(* obsolete support after version 2.7.0.1
-------------------------read the document bellow---------------------------------------------------------------*)
FUNCTION_BLOCK FB_IPRO_ModbusRTU EXTENDS FB_ModbusSlaveRtu IMPLEMENTS I_Ipro_MotorPower;
VAR
	eState : E_AxisState;
// Write Modbus
	bControlModeSwitchCommand	: BOOL;						(* write p4.15 *)
	bFieldbusEnableServoCommand	:  BOOL;					(* write p4.11 0:Disable, 1:Anable *)
	eControlMode : E_IProCtrlMode;
	lrPositivePositionSoftwareLimit : LREAL;
	lrNagativePositionSoftwareLimit	: LREAL;
	lrMaxSpeedLimitOfControlModeSwitch : LREAL := 100;		(* P0.90 Add:1180 :Set the max. running speed during positioning when switching from speed mode or torque mode to position mode under position/speed, position/torque compound mode.*)
	lrPositionCmd : LREAL;									(* p4.12 Position value unit:(10000/rotary) *)
	lrSpeedCmd : LREAL;										(* p4.13 Unit:(rotary/minute) *)
	lrTorqueCmd	: LREAL; 									(* p4.14 Unit:% *)
	lrMaxSpeed	: LREAL; 									(* p4.31 Unit:(rotary/minute) *)
	lrMaxTorque	: LREAL; 									(* p0.10 Unit:% *) 
	bEmergenCyStop : BOOL;									(* p4.23 add:1846 16 bit :If P4.10 is 1, this parameter can be used to set emergency stop command. *)
	
// Read modbus
	lrSpeedFeedback	: LREAL;								(* r0.00 *) 
	lrTorqueFeedback : LREAL;								(* r0.06 *)
	lrPositionFeedback : LREAL;								(* r0.02 *)
	nFaultCode : INT; 										(* r0.99 *)
	eSystemStatus : E_IProStatus; 							(* r0.30 *)
	eCurrentMode : E_IProCurrentMode ;						(* r0.32 0: Position mode, 1: speed mode, 2: torque Mode*) 
							
	TempData_Word2real : U_Word2Real;
	TempData_Word2Dint	: U_Word2Dint;
	TempData_Word2Int	: U_Word2Int;

// State Handing
	bInit: BOOL;
	bHome: BOOL;
	bBusy: BOOL;
	bMoveAbsolute: BOOL;
	bReset: BOOL;
	bMoveTorque: BOOL;
	bStopped: BOOL; 						// StopDone
	bStop: BOOL;							// StopRequest
	lrHomePosition: LREAL;
	bHomed: BOOL;							// home done
	bInited: BOOL;							// Init Done
	bMoveAbsoluted: BOOL;					// MoveAbs Done
	bMoveTorqued: BOOL;						// MoveTorque Done
	bAbort: BOOL;							// Abort Request
	bActive: BOOL;
END_VAR

(*-------------------Document-------------
	1 set param in drive soft
	2 if set the control mode is different than Curren control mode on the Drive, The drive need restart by drive soft OR turn off power
	3 if the control mode swith command is TRUE, the current control mode will change according to the second mode if eControlMode have
	for example eControlMode = PositionTorque, when bControlModeSwitchCommand = false , currentmode is Position, else current mode is torque if it can
*)

bActive := eState >= AXIS_READY_INITIALIZED;
StateMachine();
bError := nFaultCode <> 0;
SUPER^();
CASE eState OF
	AXIS_INITIALIZING..AXIS_RESET_DONE, AXIS_ABORTING:
		tonConfirmReallyError(
			IN := bError OR bModbusError,
			PT := timeConfirmReallyError,
			Q => bReallyError 
		);
END_CASE

PROPERTY Active : bool
GET
Active := bActive;
END_GET
END_PROPERTY

{attribute 'monitoring' := 'variable'}
PROPERTY Busy : bool
GET
Busy := bBusy;
END_GET
END_PROPERTY

PROPERTY ControlMode : E_IProCtrlMode
GET
END_GET
SET
IF eState = AXIS_UNINITIALIZED THEN
	THIS^.eControlMode := ControlMode;
END_IF
END_SET
END_PROPERTY

PROPERTY ControlModeSwitchCmd : bool
GET
ControlModeSwitchCmd := bControlModeSwitchCommand;
END_GET
END_PROPERTY

METHOD Convert : BOOL
VAR_INPUT
	iRegionNo	:	INT;
	pReadData	:	POINTER TO word;
END_VAR
VAR
	iLoop		: 	INT;
	TempData	:	 U_Word2Dint;
	TempData_w2i	: U_Word2Int;
	TempData_Int	: INT;
END_VAR
	TempData.iWord[0] := pReadData[0];
	TempData.iWord[1] := pReadData[1];
	TempData_w2i.iWord := pReadData[0];
	TempData_Int := TempData_w2i.iInt;
CASE iRegionNo OF 
	0:// speed 0.1 r/m
		lrSpeedFeedback := DINT_TO_LREAL(TempData.idInt)*0.1;//32 bit
	1:// position unit 1
	
		lrPositionFeedback := DINT_TO_LREAL(TempData.idInt); //64 bit
	2:// torque 0.1
		lrTorqueFeedback := INT_TO_LREAL(TempData_Int)*0.1;
	3:
		eSystemStatus := pReadData[0];
	4:
		eCurrentMode := pReadData[0];
	5:
		nFaultCode := pReadData[0];// must not use word to int

	
END_CASE
END_METHOD

PROPERTY CurrentMode : E_IProCurrentMode
GET
CurrentMode := eCurrentMode;
END_GET
END_PROPERTY

PROPERTY Enable : bool
GET
Enable := bFieldbusEnableServoCommand;
END_GET
END_PROPERTY

PROPERTY ErrorID : REFERENCE TO INT
GET
ErrorID REF= nFaultCode;
END_GET
END_PROPERTY

{attribute 'monitoring' := 'variable'}
PROPERTY InPosition : bool
GET
InPosition := F_CheckInRange( lrHighLimit := lrPositionFeedback + 20,
						lrLowLimit := lrPositionFeedback - 20,
						lrValue := lrPositionCmd)	;
END_GET
END_PROPERTY

PROPERTY IsHomed : bool
GET
IsHomed := F_CheckInRange( lrHighLimit := lrPositionFeedback + 10,
						lrLowLimit := lrPositionFeedback - 10,
						lrValue := lrHomePosition)	;
END_GET
END_PROPERTY

PROPERTY IsInTorque : bool
GET
isIntorque := F_CheckInRange( lrHighLimit := lrTorqueFeedback + 0.5,// 1%
					lrLowLimit := lrTorqueFeedback -0.5 ,
					lrValue := lrTorqueCmd) ;// +-0.5%	;
END_GET
END_PROPERTY

PROPERTY IsStop : bool // not moving
GET
IsStop := eSystemStatus = IPRO_STATUS_FAULT;
END_GET
END_PROPERTY

PROPERTY MaxSpeed : lreal// large than 0
GET
MaxSpeed := lrMaxSpeed;
END_GET
SET
IF eState = AXIS_UNINITIALIZED THEN
	lrMaxSpeed := MaxSpeed;
END_IF
END_SET
END_PROPERTY

PROPERTY MaxTorque : Lreal// // % larger than 0
GET
MaxTorque := lrMaxTorque;
END_GET
SET
IF eState = AXIS_UNINITIALIZED THEN
	lrMaxTorque := MaxTorque;
END_IF

arrAddressWrite[10][2] :=  LREAL_TO_WORD(ABS(lrMaxTorque*10));
END_SET
END_PROPERTY

METHOD MR_Abort : BOOL // THIS IS REQUEST ABORT. => ACTIVE = False
IF eState >= AXIS_INITIALIZING THEN
	bAbort := TRUE;
	MR_Abort := FALSE;
	bBusy := TRUE;
	eState := AXIS_ABORTING;
ELSIF eState = AXIS_UNINITIALIZED THEN
	bAbort := FALSE;
	MR_Abort := TRUE;
	bBusy := False;
END_IF
END_METHOD

METHOD MR_Home : BOOL // control mode must have Position Mode // actually it the same as MOVE absolute 
VAR_INPUT
	lrHomePosition : LREAL;
END_VAR
IF eState = AXIS_IDLE AND eCurrentMode = IPRO_CURRENT_MODE_POSITION 
AND NOT F_CheckInRange(lrHighLimit := lrHomePosition + 10,
					lrLowLimit := lrHomePosition - 10,
					lrValue := lrPositionFeedback)
THEN 
	bHome := TRUE;
	bHomed := FALSE;
	bBusy := TRUE;
	MR_Home := FALSE;
 	eState := AXIS_HOME;
	THIS^.lrHomePosition := lrHomePosition;
ELSIF  eState = AXIS_IDLE AND eCurrentMode <> IPRO_CURRENT_MODE_POSITION THEN 
	bHome := TRUE;
	bHomed := FALSE;
	bBusy := TRUE;
	MR_Home := FALSE;
 	MS_SwitchMode(eModeChangeTo := IPRO_CURRENT_MODE_POSITION);

ELSIF eState = AXIS_HOME_DONE THEN
	bHomed := TRUE;
	bHome := FALSE;
	bBusy := FALSE;
	MR_Home := TRUE;
END_IF
END_METHOD

METHOD MR_Init : BOOL
IF eState = AXIS_UNINITIALIZED THEN
	bInit := TRUE;
	bInited := FALSE;
	bBusy := TRUE;
	MR_Init := FALSE;
	eState := AXIS_INITIALIZING;
ELSIF eState = AXIS_READY_INITIALIZED THEN
	bInited := True;
	bInit := FALSE;
	bBusy := FALSE;
	MR_Init := TRUE;
	
END_IF
END_METHOD

METHOD MR_MoveAbsolute : BOOL // control mode must have Position Mode
VAR_INPUT
	lrAbsolutePosition : LREAL;
END_VAR
IF eState = AXIS_IDLE 
AND eCurrentMode = IPRO_CURRENT_MODE_POSITION 
AND NOT F_CheckInRange( lrHighLimit := lrPositionFeedback + 10,
						lrLowLimit := lrPositionFeedback - 10,
						lrValue := lrAbsolutePosition)													
THEN
	lrPositionCmd := lrAbsolutePosition;
	MR_MoveAbsolute := FALSE;
	bBusy := TRUE;
	bMoveAbsolute := TRUE;
	bMoveAbsoluted := FALSE;
	eState := AXIS_MOVE_ABSOLUTE;
ELSIF eState = AXIS_IDLE  AND eCurrentMode <> IPRO_CURRENT_MODE_POSITION THEN
	MR_MoveAbsolute := FALSE;
	bBusy := TRUE;
	bMoveAbsolute := TRUE;
	bMoveAbsoluted := FALSE;
	MS_SwitchMode( eModeChangeTo := IPRO_CURRENT_MODE_POSITION);// if switch mode ok => eCurrentMode = AXIS_CURRENT_MODE_POSITION 

ELSIF eState = AXIS_MOVE_ABSOLUTE_DONE THEN
	bBusy := FALSE;
	bMoveAbsolute := FALSE;
	MR_MoveAbsolute := TRUE;
	bMoveAbsoluted := TRUE;
	
ELSIF  eState = AXIS_IDLE 
	AND eCurrentMode = IPRO_CURRENT_MODE_POSITION 
	AND F_CheckInRange( lrHighLimit := lrPositionFeedback + 10,
							lrLowLimit := lrPositionFeedback - 10,
							lrValue := lrAbsolutePosition)													
	THEN
		bBusy := FALSE;
		bMoveAbsolute := FALSE;
		MR_MoveAbsolute := TRUE;
		bMoveAbsoluted := TRUE;
END_IF
END_METHOD

METHOD MR_MoveTorque : BOOL // control mode must have torque Mode edit :Torque can be change every time if needed;
VAR_INPUT
	lrTorque	: LREAL;// must smaller than max torque
END_VAR
IF eState = AXIS_IDLE
	AND eCurrentMode = IPRO_CURRENT_MODE_TORQUE 
	AND NOT F_CheckInRange(
				lrHighLimit := lrTorqueFeedback + 0.5,// 1%
				lrLowLimit := lrTorqueFeedback -0.5 ,
				lrValue := lrTorque) // +-0.5%	
THEN
	bMoveTorque	:= TRUE;
	bMoveTorqued	:= FALSE;
	bBusy := TRUE;
	MR_MoveTorque := FALSE;
	eState := AXIS_MOVE_TORQUE;
	lrTorqueCmd := lrTorque;
	
ELSIF eState = AXIS_IDLE
	AND eCurrentMode<>IPRO_CURRENT_MODE_TORQUE
THEN
	MR_MoveTorque := FALSE;
	bBusy := TRUE;
	bMoveTorque := TRUE;
	bMoveTorqued	:= FALSE;
	MS_SwitchMode(eModeChangeTo := IPRO_CURRENT_MODE_TORQUE);// if switch mode ok => eCurrentMode = IPRO_CURRENT_MODE_POSITION 

ELSIF eState = AXIS_IDLE 
	OR eState = AXIS_MOVE_TORQUE_DONE 
THEN
	bBusy := FALSE;
	bMoveTorque := FALSE;
	MR_MoveTorque := TRUE;
	bMoveTorqued	:= TRUE;
END_IF
END_METHOD

METHOD MR_Reset : BOOL// can't not use this method because i didn't find way to reset
(*IF eState <> IPRO_RESET AND eState <> IPRO_RESET_DONE THEN
	bReset := TRUE;
	MR_Reset := FALSE;
	eState := IPRO_RESET;
ELSIF eState = IPRO_RESET_DONE THEN
	bReset := FALSE;
	MR_Reset := TRUE;
	
END_IF*)
END_METHOD

METHOD MR_Stop : BOOL
IF eState >= AXIS_IDLE AND eState <> AXIS_STOP_DONE THEN
	bStop := TRUE;
	bStopped := FALSE;
	MR_Stop := FALSE;
	eState := AXIS_STOP;
	bBusy := TRUE;
ELSIF eState = AXIS_STOP_DONE THEN
	bStop := FALSE;
	bStopped := TRUE;
	MR_Stop := TRUE;
	bBusy := FALSE;
END_IF
END_METHOD

METHOD PROTECTED MS_Aborting// still remain all the params set before init
VAR_INPUT
END_VAR
bFieldbusEnableServoCommand := FALSE;
lrSpeedCmd := 0;
lrPositionCmd := 0;
lrTorqueCmd := 0;
bEmergenCyStop := false;
arrAddressWrite[1][2] :=  BOOL_TO_WORD(bFieldbusEnableServoCommand);
IF THIS^.eSystemStatus <> IPRO_STATUS_RUN THEN
	eState := AXIS_UNINITIALIZED;
END_IF
END_METHOD

METHOD PROTECTED MS_Home
VAR_INPUT
END_VAR
TempData_Word2Dint.idInt := LREAL_TO_DINT(lrHomePosition);
arrAddressWrite[6][2] := TempData_Word2Dint.iWord[0];
arrAddressWrite[6][3] := TempData_Word2Dint.iWord[1];

IF F_CheckInRange(lrHighLimit := lrHomePosition + 10,
					lrLowLimit := lrHomePosition - 10,
					lrValue := lrPositionFeedback)
THEN
	eState := AXIS_HOME_DONE;
END_IF
END_METHOD

METHOD PROTECTED  MS_HomeDone
VAR_INPUT
END_VAR
IF NOT bHome THEN
	eState := AXIS_IDLE;
END_IF
END_METHOD

METHOD PROTECTED MS_Idle
VAR_INPUT
END_VAR
;
END_METHOD

METHOD PROTECTED MS_Initializing
VAR_INPUT
END_VAR
// this servo can't reset error by modbus
IF THIS^.eSystemStatus = IPRO_STATUS_READY THEN // Ignor the faultcode AND nFaultCode = 0  THEN
	bFieldbusEnableServoCommand := TRUE;
	arrAddressWrite[1][2] := BOOL_TO_WORD(bFieldbusEnableServoCommand);
END_IF
 
IF eSystemStatus = IPRO_STATUS_RUN THEN
	eState := AXIS_READY_INITIALIZED;
END_IF
END_METHOD

METHOD PROTECTED MS_MoveAbsolute
VAR_INPUT
END_VAR
TempData_Word2Dint.idInt := LREAL_TO_DINT(lrPositionCmd);
arrAddressWrite[6][2] := TempData_Word2Dint.iWord[0];
arrAddressWrite[6][3] := TempData_Word2Dint.iWord[1];

IF F_CheckInRange(lrHighLimit := lrPositionCmd + 10,
					lrLowLimit := lrPositionCmd - 10,
					lrValue := lrPositionFeedback)
THEN
	eState := AXIS_MOVE_ABSOLUTE_DONE;
END_IF
END_METHOD

METHOD PROTECTED MS_MoveAbsoluteDone
VAR_INPUT
END_VAR
IF NOT bMoveAbsolute THEN
	eState := AXIS_IDLE;
END_IF
END_METHOD

METHOD PROTECTED MS_MoveTorque
VAR_INPUT
END_VAR
TempData_Word2Int.iInt := LREAL_TO_INT(lrTorqueCmd *10);
arrAddressWrite[8][2] :=  TempData_Word2Int.iWord;
(* should by pass this one if not, it can't receive new Torque
IF F_CheckInRange( lrHighLimit := lrTorqueFeedback + 0.5,// 1%
					lrLowLimit := lrTorqueFeedback -0.5 ,
					lrValue := lrTorqueCmd) 
THEN
	eState := IPRO_MOVE_TORQUE_DONE;
END_IF*)
eState := AXIS_MOVE_TORQUE_DONE;
END_METHOD

METHOD PROTECTED MS_MoveTorqueDone
VAR_INPUT
END_VAR
IF NOT bMoveTorque THEN
	eState := AXIS_IDLE;
END_IF
END_METHOD

METHOD PROTECTED MS_ReadyInitialized
VAR_INPUT
END_VAR
IF NOT bInit THEN
	eState := AXIS_IDLE;
END_IF
END_METHOD

METHOD PROTECTED MS_Reset
VAR_INPUT
END_VAR
END_METHOD

METHOD PROTECTED MS_ResetDone
VAR_INPUT
END_VAR
END_METHOD

METHOD PROTECTED MS_Stop
VAR_INPUT
END_VAR
bEmergenCyStop := TRUE;
arrAddressWrite[11][2] := BOOL_TO_WORD(THIS^.bEmergenCyStop);
IF eSystemStatus = IPRO_STATUS_FAULT THEN
	eState := AXIS_STOP_DONE;
END_IF
END_METHOD

METHOD PROTECTED MS_StopDone
VAR_INPUT
END_VAR
IF NOT bStop THEN
	eState := AXIS_UNINITIALIZED;
END_IF
END_METHOD

METHOD PROTECTED MS_SwitchMode : BOOL;
VAR_INPUT
	eModeChangeTo	: E_IProCurrentMode; // False is the first mode , TRUE is Seconde Mode in Control mode
END_VAR


CASE THIS^.eControlMode OF
	
	IPRO_CTRL_MODE_POSITION_TORQUE:
		IF eModeChangeTo = IPRO_CURRENT_MODE_POSITION THEN
			bControlModeSwitchCommand := FALSE;
		ELSIF eModeChangeTo = IPRO_CURRENT_MODE_TORQUE THEN
			bControlModeSwitchCommand := TRUE;
		END_IF
	IPRO_CTRL_MODE_POSITION_SPEED:
		IF eModeChangeTo = IPRO_CURRENT_MODE_POSITION THEN
			bControlModeSwitchCommand := FALSE;
		ELSIF eModeChangeTo = IPRO_CURRENT_MODE_SPEED THEN
			bControlModeSwitchCommand := TRUE;
		END_IF
	IPRO_CTRL_MODE_SPEED_TORQUE:
		IF eModeChangeTo = IPRO_CURRENT_MODE_SPEED THEN
			bControlModeSwitchCommand := FALSE;
		ELSIF eModeChangeTo = IPRO_CURRENT_MODE_TORQUE THEN
			bControlModeSwitchCommand := TRUE;
		END_IF
	
END_CASE

arrAddressWrite[0][2] :=  BOOL_TO_WORD(bControlModeSwitchCommand); 

IF eCurrentMode = eModeChangeTo THEN
	MS_SwitchMode := TRUE;
ELSE
	MS_SwitchMode := FALSE;	
END_IF
END_METHOD

METHOD PROTECTED MS_Uninitalized
VAR_INPUT
END_VAR
bBusy := FALSE;
arrAddressRead[0][0] := 4000;// motor speed FB //0.1 r/min // 4000, 4001
arrAddressRead[0][1] := 2;
arrAddressRead[0][2] := E_ModbusFunction.ReadHoldingRegisters;

arrAddressRead[1][0] := 4004;// motor position FB// reference unit 
arrAddressRead[1][1] := 4;
arrAddressRead[1][2] := E_ModbusFunction.ReadHoldingRegisters;

arrAddressRead[2][0] := 4016;// motor Torque FB// reference unit 
arrAddressRead[2][1] := 1;
arrAddressRead[2][2] := E_ModbusFunction.ReadHoldingRegisters;

arrAddressRead[3][0] := 4064;// System status // 
arrAddressRead[3][1] := 1;
arrAddressRead[3][2] := E_ModbusFunction.ReadHoldingRegisters;

arrAddressRead[4][0] := 4068;// Current Mode 
arrAddressRead[4][1] := 1;
arrAddressRead[4][2] := E_ModbusFunction.ReadHoldingRegisters;

arrAddressRead[5][0] := 4198;// FaultCode
arrAddressRead[5][1] := 1;
arrAddressRead[5][2] := E_ModbusFunction.ReadHoldingRegisters;	
iNumAddRegionRead := 6;
// write
arrAddressWrite[0][0] := 1830;// 
arrAddressWrite[0][1] := 1;
arrAddressWrite[0][2] := BOOL_TO_WORD(bControlModeSwitchCommand); // disable first
arrAddressWrite[0][10]	:= E_ModbusFunction.WriteSingleRegister;

arrAddressWrite[1][0] := 1822;// 
arrAddressWrite[1][1] := 1;
arrAddressWrite[1][2] :=  BOOL_TO_WORD(bFieldbusEnableServoCommand); // disable first
arrAddressWrite[1][10] := E_ModbusFunction.WriteSingleRegister;

arrAddressWrite[2][0] := 1006;// 
arrAddressWrite[2][1] := 1;
arrAddressWrite[2][2] := eControlMode; 
arrAddressWrite[2][10] := E_ModbusFunction.WriteSingleRegister;

arrAddressWrite[3][0] := 1070;//  //32 bit 1070, 1071
arrAddressWrite[3][1] := 2;
TempData_Word2Dint.idInt := LREAL_TO_DINT(lrPositivePositionSoftwareLimit);
arrAddressWrite[3][2] := TempData_Word2Dint.iWord[0];
arrAddressWrite[3][3] := TempData_Word2Dint.iWord[1];
arrAddressWrite[3][10] := E_ModbusFunction.WriteMultipleRegisters;

arrAddressWrite[4][0] := 1072;//  //32 bit 1072, 1073
arrAddressWrite[4][1] := 2;
TempData_Word2Dint.idInt := LREAL_TO_DINT(lrNagativePositionSoftwareLimit);
arrAddressWrite[4][2] := TempData_Word2Dint.iWord[0];
arrAddressWrite[4][3] := TempData_Word2Dint.iWord[1];
arrAddressWrite[4][10] := E_ModbusFunction.WriteMultipleRegisters;

arrAddressWrite[5][0] := 1180;// 
arrAddressWrite[5][1] := 1;
arrAddressWrite[5][2] :=  LREAL_TO_WORD(lrMaxSpeedLimitOfControlModeSwitch); 
arrAddressWrite[5][10] := E_ModbusFunction.WriteSingleRegister;

arrAddressWrite[6][0] := 1824;// 32 bit 1825
arrAddressWrite[6][1] := 2;
TempData_Word2Dint.idInt := LREAL_TO_DINT(lrPositionCmd);
arrAddressWrite[6][2] := TempData_Word2Dint.iWord[0];
arrAddressWrite[6][3] := TempData_Word2Dint.iWord[1];
arrAddressWrite[6][10] := E_ModbusFunction.WriteMultipleRegisters;

arrAddressWrite[7][0] := 1826;//16 bit
arrAddressWrite[7][1] := 1;
TempData_Word2Int.iInt := LREAL_TO_INT(lrSpeedCmd);
arrAddressWrite[7][2] :=  TempData_Word2Int.iWord;
arrAddressWrite[7][10] := E_ModbusFunction.WriteSingleRegister;

arrAddressWrite[8][0] := 1828;// 16 bit
arrAddressWrite[8][1] := 1;
TempData_Word2Int.iInt := LREAL_TO_INT(lrTorqueCmd);
arrAddressWrite[8][2] :=  TempData_Word2Int.iWord;
arrAddressWrite[8][10] := E_ModbusFunction.WriteSingleRegister;

arrAddressWrite[9][0] := 1862;// 1
arrAddressWrite[9][1] := 1;
TempData_Word2Int.iInt := LREAL_TO_INT(ABS(lrMaxSpeed));
arrAddressWrite[9][2] := TempData_Word2Int.iWord;
arrAddressWrite[9][10] := E_ModbusFunction.WriteSingleRegister;

arrAddressWrite[10][0] := 1020;// 32 bit 1825/ //0.1 PERCENT
arrAddressWrite[10][1] := 1;
arrAddressWrite[10][2] := LREAL_TO_WORD(ABS(lrMaxTorque*10));
arrAddressWrite[10][10]	:= E_ModbusFunction.WriteSingleRegister;

arrAddressWrite[11][0] := 1846;
arrAddressWrite[11][1] := 1;
arrAddressWrite[11][2] := BOOL_TO_WORD(THIS^.bEmergenCyStop);
arrAddressWrite[11][10]	:= E_ModbusFunction.WriteSingleRegister;
iNumAddRegionWrite := 12;
END_METHOD

PROPERTY NagativePositionLimit : lreal
GET
NagativePositionLimit := lrNagativePositionSoftwareLimit;
END_GET
SET
IF eState = AXIS_UNINITIALIZED THEN
	lrNagativePositionSoftwareLimit := NagativePositionLimit;
END_IF
END_SET
END_PROPERTY

PROPERTY PositionCmd : lreal
GET
PositionCmd := lrPositionCmd;
END_GET
END_PROPERTY

PROPERTY PositionFeedBack : lreal
GET
PositionFeedBack := lrPositionFeedback;
END_GET
END_PROPERTY

PROPERTY PositionPositiveLimit : lreal
GET
PositionPositiveLimit := lrPositivePositionSoftwareLimit;
END_GET
SET
IF eState = AXIS_UNINITIALIZED THEN
	lrPositivePositionSoftwareLimit := PositionPositiveLimit;
END_IF
END_SET
END_PROPERTY

PROPERTY ReallyError : bool
SET
ReallyError := bReallyError;
END_SET
END_PROPERTY

PROPERTY SpeedCmd : LREAL // r/ minute
GET
SpeedCmd := lrSpeedCmd;
END_GET
SET
lrSpeedCmd := SpeedCmd;
TempData_Word2Int.iInt := LREAL_TO_INT(lrSpeedCmd*10);
arrAddressWrite[7][2] :=  TempData_Word2Int.iWord;
END_SET
END_PROPERTY

PROPERTY SpeedFeedback : Lreal
GET
SpeedFeedback := lrSpeedFeedback;
END_GET
END_PROPERTY

PROPERTY State : E_AxisState
GET
State := eState;
END_GET
END_PROPERTY

METHOD PROTECTED StateMachine
VAR_INPUT
END_VAR

VAR

END_VAR
CASE eState OF
	AXIS_UNINITIALIZED:
		MS_Uninitalized();
		
	AXIS_INITIALIZING:
		MS_Initializing();
		
	AXIS_READY_INITIALIZED:
		MS_ReadyInitialized();
		
	AXIS_IDLE:
		MS_Idle();
		
	AXIS_HOME:
		MS_Home();
		
	AXIS_HOME_DONE:
		MS_HomeDone();
		
	AXIS_MOVE_ABSOLUTE:
		MS_MoveAbsolute();
	
	AXIS_MOVE_ABSOLUTE_DONE:
		MS_MoveAbsoluteDone();
		
	AXIS_MOVE_TORQUE:
		MS_MoveTorque();
		
	AXIS_MOVE_TORQUE_DONE: 
		MS_MoveTorqueDone();
	
	AXIS_STOP:
		MS_Stop();
	
	AXIS_STOP_DONE:
		MS_StopDone();
		
	AXIS_RESET:
		MS_Reset();
	
	AXIS_RESET_DONE:
		MS_ResetDone();
		
	AXIS_ABORTING:
		MS_Aborting();
	

		
END_CASE
END_METHOD

PROPERTY Status : E_IProStatus
GET
Status := eSystemStatus;
END_GET
END_PROPERTY

PROPERTY TorqueCmd : lreal // %
GET
TorqueCmd :=  lrTorqueCmd ;
END_GET
END_PROPERTY

PROPERTY TorqueFeedback : lreal
GET
TorqueFeedback := lrTorqueFeedback;
END_GET
END_PROPERTY

END_FUNCTION_BLOCK

(* stored: Version 1.1.0.1, ProductVersion 3.1.4024.12
   POU FB_IPRO_ModbusRTU: Id {779a38f8-03a4-4a78-bdd8-18318bba4a44}, SpecialFunc None
   Folder Parameters: Id {135f1342-f3ac-470e-b188-26cd0d7b27c7}
   Folder parent: Id {6b07bf69-3a52-4263-9762-d97c1b99a02c}
   Folder Requests: Id {fab6c147-feaf-4bd7-9ed7-49433b01dc12}
   Folder SetBeforInit: Id {f9ae4f66-d74b-40ad-8929-ca4d65a2caf5}
   Folder StateMachine: Id {bc03708e-6405-480e-aa24-527bc8f89ef2}
   Folder Status: Id {40a08b4a-5fb9-44d8-be2c-031269a557ba}
   Property Active: Id {b4a9866b-0d33-4922-95c7-beca9bac3388}
   Get Get: Id {78e8bb07-e221-4b68-8e28-09652440fb31}
   Property Busy: Id {04fd7b58-cd07-4eba-8564-70318006a4ac}
   Get Get: Id {4c84cee3-c2c5-4fe5-9f67-ec059c453e7a}
   Property ControlMode: Id {82f3a655-7191-41d9-b3e9-013c4502fd03}
   Get Get: Id {f24d0a22-b23c-4e93-b024-b2cd29a0591e}
   Set Set: Id {fac56fc0-c696-47ae-b960-e57bcfe47507}
   Property ControlModeSwitchCmd: Id {a97f4de7-79f1-4a8b-aeb0-fb6d46c8368c}
   Get Get: Id {fa8c8626-2fdf-4d50-9d7b-b003da3c03a4}
   Method Convert: Id {a0f2c8db-6069-46f2-b7e6-10beb6b999d1}
   Property CurrentMode: Id {d11bf5fa-8718-44ad-8a77-3f70675bc099}
   Get Get: Id {0142fdff-63a5-4bb1-b024-753ebd04f18c}
   Property Enable: Id {855be6cb-afa6-4670-b51a-ed92bd24485e}
   Get Get: Id {1487b77a-cc23-4513-8843-d56b811200cd}
   Property ErrorID: Id {0b249e37-0a65-4ec1-a1e6-71c97f90b6db}
   Get Get: Id {0e3d4b6a-993d-4a39-b37f-82be1b4cd517}
   Property InPosition: Id {4ad81687-b948-4488-aa5b-2ac52454fe3d}
   Get Get: Id {cafeb194-f541-43df-9a96-6fa2f21aa8ce}
   Property IsHomed: Id {25150335-f115-450b-8103-c4c59b87dcd8}
   Get Get: Id {2d3d439b-5162-456e-97d7-e2931abe5269}
   Property IsInTorque: Id {5cc895c7-6ab9-4745-bbf3-251c0a00b39b}
   Get Get: Id {3e20b4a0-b649-4f36-97c9-bad969a3fe7d}
   Property IsStop: Id {721186bc-60dd-4115-8523-deb6a9e576b6}
   Get Get: Id {8a4cae79-0c89-49af-94e4-a422fbdbcc15}
   Property MaxSpeed: Id {efa9fab6-f7e3-406f-adb2-b575f7b68621}
   Get Get: Id {7a42f7f8-ceb6-4e59-88ef-de6a9a2782d1}
   Set Set: Id {ef5b532c-d4c2-4431-917a-6cd0d488cedb}
   Property MaxTorque: Id {8197c65c-569c-4655-9971-34203364c4a1}
   Get Get: Id {1222d17e-9006-4bc5-910b-dd7509f7de1e}
   Set Set: Id {9a3480e6-a1ae-4445-be64-e3d7fd6f3a0c}
   Method MR_Abort: Id {c01a224b-502a-4fb8-86bb-578474547fce}
   Method MR_Home: Id {0bedcd25-5802-4be5-b446-f54e355f5942}
   Method MR_Init: Id {bdf0da52-3dbd-43dd-b4d0-dd24e17ac0ad}
   Method MR_MoveAbsolute: Id {ca744ba7-f549-4cdc-bd1f-573625e34a4f}
   Method MR_MoveTorque: Id {0d0a9f5b-f53f-4d27-b09a-5da162d32222}
   Method MR_Reset: Id {2b2c7fb3-bf71-451a-9128-c4cbe2a3c533}
   Method MR_Stop: Id {4b80d5e7-5616-4415-8bd0-c2a744c8ce87}
   Method MS_Aborting: Id {6669002e-7ddc-4f29-b09d-fa81ccb85f53}
   Method MS_Home: Id {a82686d0-19c1-4705-8230-910afbff76c7}
   Method MS_HomeDone: Id {8c5d1efa-8d28-4f3a-988f-d958eaca4b42}
   Method MS_Idle: Id {8858a3c4-b1ef-4e3d-9003-fec5be52e4f5}
   Method MS_Initializing: Id {54c9912c-a57e-47b7-9c2e-cde4ab36bc1f}
   Method MS_MoveAbsolute: Id {b775430d-4bdd-45a4-a486-584aacedb928}
   Method MS_MoveAbsoluteDone: Id {c8076e55-0cd3-419b-915d-ba528fd9900e}
   Method MS_MoveTorque: Id {1f758174-9816-41b3-b0c1-93e4728f4c89}
   Method MS_MoveTorqueDone: Id {8f9b48d7-1fdb-40bd-8df1-6de155336372}
   Method MS_ReadyInitialized: Id {cbc8a9ef-9949-4a0d-8ef9-e49466e0046c}
   Method MS_Reset: Id {a9cc5e5b-bbec-41b9-b69b-a7457e556196}
   Method MS_ResetDone: Id {f08aa95a-6a54-4ffd-b94a-dcc9c286e2a9}
   Method MS_Stop: Id {f30ba650-5154-4e65-b042-d8ef3dc35992}
   Method MS_StopDone: Id {9ad74a08-b438-4ff2-acef-4f3b29d4b54f}
   Method MS_SwitchMode: Id {40b3eeee-e744-4506-b2ff-c6859ef0c1b9}
   Method MS_Uninitalized: Id {c0b072b8-11b2-49e7-943c-d6804dcfcc94}
   Property NagativePositionLimit: Id {a1a1c3fa-f229-4e2d-9766-ec703c2de587}
   Get Get: Id {c561b735-862d-4dab-85ab-1ac0a4668272}
   Set Set: Id {f60d0a52-4490-4908-8f23-4e565feffa59}
   Property PositionCmd: Id {23e83466-f96c-4622-876f-5a6f8b31225b}
   Get Get: Id {4ffc8f22-a5cd-40fb-ac2c-b551154bd191}
   Property PositionFeedBack: Id {f1fa1bdb-f57d-44eb-ae97-8f48f67d5f70}
   Get Get: Id {00164334-2f50-4d35-9dd2-0ed5521dba27}
   Property PositionPositiveLimit: Id {06450a26-3ac9-492f-8bb9-df1b1a771fb7}
   Get Get: Id {33877c33-0487-4a3c-ad63-fd496fe84bd7}
   Set Set: Id {900ac512-6122-4a49-8d3e-903adf79f440}
   Property ReallyError: Id {131e458f-64bc-44a3-a841-415854b490d0}
   Set Set: Id {15d805cb-fa21-450c-8426-92b4717cf052}
   Property SpeedCmd: Id {0a3d1347-d85b-4fe3-ba98-003bcfd016d4}
   Get Get: Id {ff03e774-b178-46dd-98e1-0a1339fb2aca}
   Set Set: Id {f22aed52-55fa-44fd-adb4-6e7498b50529}
   Property SpeedFeedback: Id {8c0c65e8-744a-4ad5-a009-67c9db3f6e5a}
   Get Get: Id {364a84ad-39b8-4928-b5bb-abe5794f9595}
   Property State: Id {ca3be74d-8a42-48c3-bc02-f193a7afc1dd}
   Get Get: Id {34666fd9-328f-4f91-a8b2-ddcc78b6d879}
   Method StateMachine: Id {8d3ffbfd-6d5e-4328-9d69-29932a291b26}
   Property Status: Id {945903a2-3273-4225-9050-43cbdf878bdb}
   Get Get: Id {d6f6803a-14f1-44f6-b590-ec4070c2bb8a}
   Property TorqueCmd: Id {fc7bc3e0-4bca-41e7-a5ee-2bbc532aa88e}
   Get Get: Id {9b9e5f35-2aeb-4fe1-bf67-9fdf730cacc9}
   Property TorqueFeedback: Id {f47dfc44-d2a1-41d7-a3ca-f94ced010654}
   Get Get: Id {41d90d48-da2f-46b1-b277-8d115eea513d} *)
